Fanuc KAREL source: compact_preamble.KL

PROGRAM KF00072
%NOLOCKGROUP
VAR
I:INTEGER;J:INTEGER;X:REAL;Y:REAL;B:BOOLEAN;C:BOOLEAN;TXT : STRING[80];TXT2 : STRING[80];AI : ARRAY[4] OF INTEGER;BI : ARRAY[4] OF INTEGER;P : XYZWPR
JP : JOINTPOS9
PF : POSITION
V1 : VECTOR
V2 : VECTOR
STATUS:INTEGER
BEGIN
TXT='12'
TXT2='2'
I=12
X=2.5
TXT2=SUB_STR(TXT,2,2)
END KF00072
